// TIA Portal V15.1 export
// export: Created 2024-06-21T08:40:52.9908373Z, ExportSetting WithDefaults, DisplayName Totally Integrated Automation Portal, DisplayVersion V15.1 Update 5, DisplayName TIA Portal Openness, DisplayVersion V15.1 Update 5, DisplayName SINAMICS Startdrive Advanced, DisplayVersion V15.1, DisplayName G130, G150, S120, S150, SINAMICS MV, S210, DisplayVersion V15.1, DisplayName G110M, G120, G120C, G120D, G120P, DisplayVersion V15.1, DisplayName STEP 7 Professional, DisplayVersion V15.1 Update 5, DisplayName STEP 7 Safety, DisplayVersion V15.1, DisplayName WinCC Professional, DisplayVersion V15.1 Update 5, DisplayName SIMATIC Visualization Architect, DisplayVersion V15.1
FUNCTION_BLOCK "L1SignalHmi"   // FB1106, FBD
TITLE = L1SignalHmi
{ S7_Optimized_Access := 'FALSE' }
AUTHOR : VCT
FAMILY : VCT
NAME : L1SigHMI
VERSION : 1.0
// ===============================================================================
// This module handles the HMI functions for one signal
// ===============================================================================
// stored: AutoNumber false, IsIECCheckEnabled false, SetENOAutomatically False, UDAEnableTagReadback false
   VAR_INPUT
      I_Signal { ExternalAccessible := 'False'; ExternalVisible := 'False'; ExternalWritable := 'False'} : Bool;   // The signal
      I_SignalCheckOn { ExternalAccessible := 'False'; ExternalVisible := 'False'; ExternalWritable := 'False'} : Bool;   // Check signal is on
      I_SignalCheckOff { ExternalAccessible := 'False'; ExternalVisible := 'False'; ExternalWritable := 'False'} : Bool;   // Check signal is off
      I_EnableAlarm { ExternalAccessible := 'False'; ExternalVisible := 'False'; ExternalWritable := 'False'} : Bool;   // Enable alarms
      I_AlarmResetPB { ExternalAccessible := 'False'; ExternalVisible := 'False'; ExternalWritable := 'False'} : Bool;   // Alarm reset pushbutton is activated
   END_VAR
   VAR_OUTPUT
      O_SignalOn { ExternalAccessible := 'False'; ExternalVisible := 'False'; ExternalWritable := 'False'} : Bool;   // Detection signal to use in program
      O_SignalAlmReqOn { ExternalAccessible := 'False'; ExternalVisible := 'False'; ExternalWritable := 'False'} : Bool;   // Request on alarm
      O_SignalAlmReqOff { ExternalAccessible := 'False'; ExternalVisible := 'False'; ExternalWritable := 'False'} : Bool;   // Request off alarm
      O_AlarmABCondition { ExternalAccessible := 'False'; ExternalVisible := 'False'; ExternalWritable := 'False'} : Bool;   // Alarm AB condition
      H_IAnim { ExternalAccessible := 'False'; ExternalVisible := 'False'; ExternalWritable := 'False'} : Word;   // For animation of the icon
   END_VAR
   VAR DB_SPECIFIC
      H_Out : Struct   // HMI
         Anim : Word;   // HMI Animation of the object
      END_STRUCT;
      SignalCheckOnAlarm { ExternalAccessible := 'False'; ExternalVisible := 'False'; ExternalWritable := 'False'} : Bool;   // Detection is not on
      SignalCheckOffAlarm { ExternalAccessible := 'False'; ExternalVisible := 'False'; ExternalWritable := 'False'} : Bool;   // Detection is not off
      AlarmCondReqOn { ExternalAccessible := 'False'; ExternalVisible := 'False'; ExternalWritable := 'False'} : Bool;   // Alarm condition
      AlarmCondReqOff { ExternalAccessible := 'False'; ExternalVisible := 'False'; ExternalWritable := 'False'} : Bool;   // Alarm condition
   END_VAR
BEGIN

REGION Network 1: **** 2.2 - Alarms - Alarm generation **** Condition alarm for active signal
   // Condition alarm for active signal
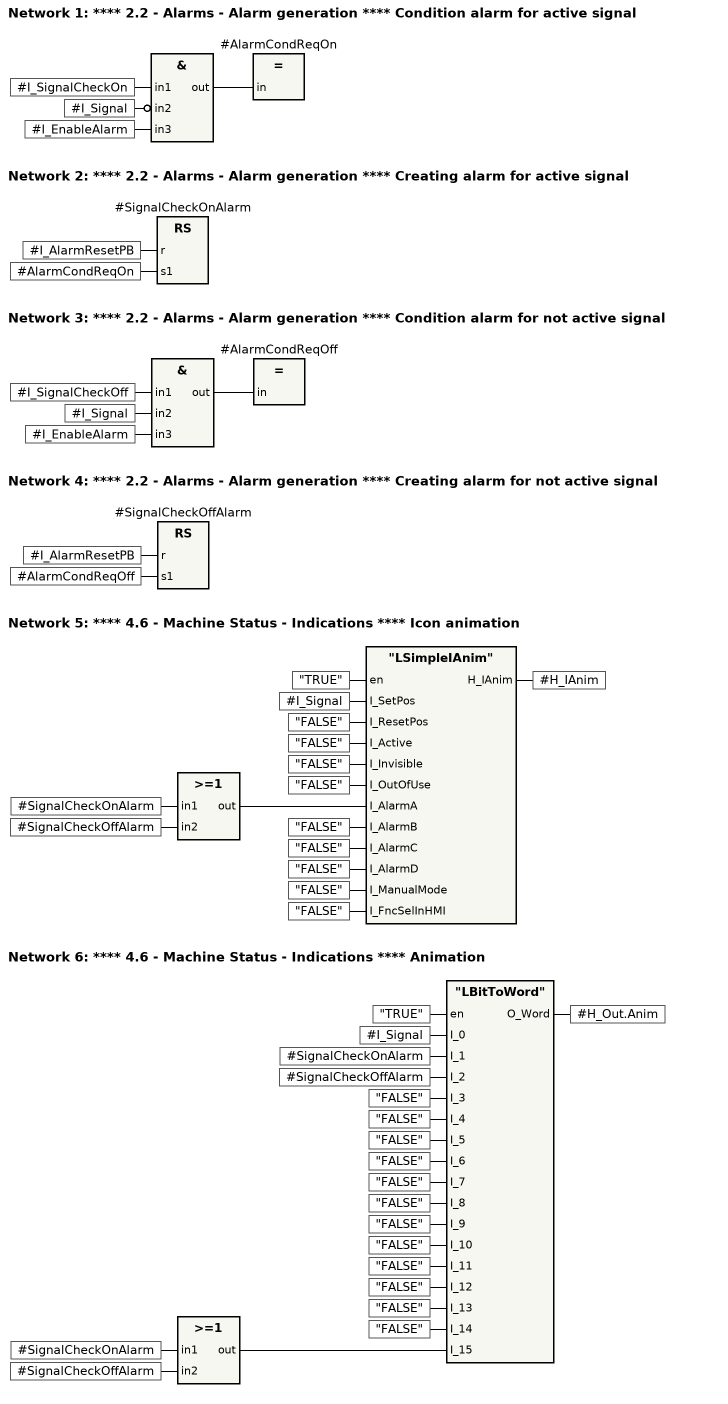
   #AlarmCondReqOn := #I_SignalCheckOn AND NOT #I_Signal AND #I_EnableAlarm;
END_REGION

REGION Network 2: **** 2.2 - Alarms - Alarm generation **** Creating alarm for active signal
   // Creating alarm for active signal
   IF #I_AlarmResetPB THEN
       #SignalCheckOnAlarm := FALSE;   // RS flip-flop
   END_IF;
   IF #AlarmCondReqOn THEN #SignalCheckOnAlarm := TRUE; END_IF;
END_REGION

REGION Network 3: **** 2.2 - Alarms - Alarm generation **** Condition alarm for not active signal
   // Condition alarm for not active signal
   #AlarmCondReqOff := #I_SignalCheckOff AND #I_Signal AND #I_EnableAlarm;
END_REGION

REGION Network 4: **** 2.2 - Alarms - Alarm generation **** Creating alarm for not active signal
   // Creating alarm for not active signal
   IF #I_AlarmResetPB THEN
       #SignalCheckOffAlarm := FALSE;   // RS flip-flop
   END_IF;
   IF #AlarmCondReqOff THEN #SignalCheckOffAlarm := TRUE; END_IF;
END_REGION

REGION Network 5: **** 4.6 - Machine Status - Indications **** Icon animation
   // Icon animation
   IF "TRUE" THEN
       "LSimpleIAnim"(I_SetPos := #I_Signal,
                      I_ResetPos := "FALSE",
                      I_Active := "FALSE",
                      I_Invisible := "FALSE",
                      I_OutOfUse := "FALSE",
                      I_AlarmA := #SignalCheckOnAlarm OR #SignalCheckOffAlarm,
                      I_AlarmB := "FALSE",
                      I_AlarmC := "FALSE",
                      I_AlarmD := "FALSE",
                      I_ManualMode := "FALSE",
                      I_FncSelInHMI := "FALSE",
                      H_IAnim => #H_IAnim);
   END_IF;
END_REGION

REGION Network 6: **** 4.6 - Machine Status - Indications **** Animation
   // Animation
   IF "TRUE" THEN
       "LBitToWord"(I_0 := #I_Signal,
                    I_1 := #SignalCheckOnAlarm,
                    I_2 := #SignalCheckOffAlarm,
                    I_3 := "FALSE",
                    I_4 := "FALSE",
                    I_5 := "FALSE",
                    I_6 := "FALSE",
                    I_7 := "FALSE",
                    I_8 := "FALSE",
                    I_9 := "FALSE",
                    I_10 := "FALSE",
                    I_11 := "FALSE",
                    I_12 := "FALSE",
                    I_13 := "FALSE",
                    I_14 := "FALSE",
                    I_15 := #SignalCheckOnAlarm OR #SignalCheckOffAlarm,
                    O_Word => #H_Out.Anim);
   END_IF;
END_REGION

REGION Network 7: *** 8 - Outputs ***** Signal on
   // Signal on
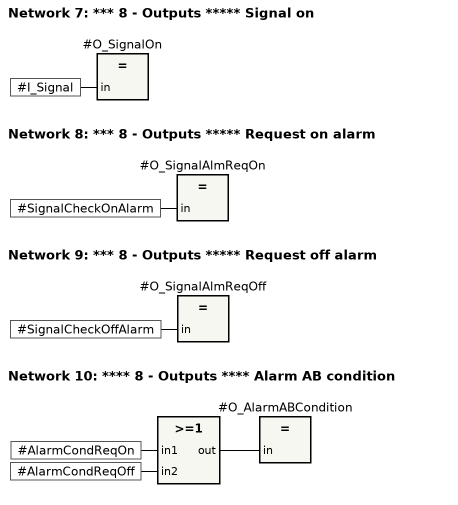
   #O_SignalOn := #I_Signal;
END_REGION

REGION Network 8: *** 8 - Outputs ***** Request on alarm
   // Request on alarm
   #O_SignalAlmReqOn := #SignalCheckOnAlarm;
END_REGION

REGION Network 9: *** 8 - Outputs ***** Request off alarm
   // Request off alarm
   #O_SignalAlmReqOff := #SignalCheckOffAlarm;
END_REGION

REGION Network 10: **** 8 - Outputs **** Alarm AB condition
   // Alarm AB condition
   #O_AlarmABCondition := #AlarmCondReqOn OR #AlarmCondReqOff;
END_REGION
END_FUNCTION_BLOCK
